VISUALIZATION _VISU_MarkViewMini  // 10x10
VAR_IN_OUT
	mInst : ST_MarkDefinition;
END_VAR
    RoundedRectangle (0,0 10x10), "%d", text variable: mInst.nId, invisible if: NOT mInst.sView.bShow, colour variable: mInst.sView.colorFill
        p3560616238: mInst.sView.nXPosPx
        p2738717112: mInst.sView.nYPosPx
END_VISUALIZATION

(* stored: Version 1.1.0.1, ProductVersion 3.1.4024.11
   Visu _VISU_MarkViewMini: Id {dbbd091e-1a3c-406d-b4ba-52ff3e22f7a8} *)
